// TIA Portal V18 export
FUNCTION_BLOCK "Pallets_Transport_System"   // FB9, LAD
{ S7_Optimized_Access := 'TRUE' }
// stored: MemoryReserve 100, SetENOAutomatically false
   VAR
      NumberOfPallet { S7_SetPoint := 'True'} : Int;
      Map : Array[1..4, 1..12] of Bool;
      MoveDirection : Int;   // 1-L, 2-Up, 3-R, 4-Down
      FoundSelectedPallet : Bool;
      CanMove : Bool;
   END_VAR
   VAR_TEMP
      i : Int;
      j : Int;
      k : Int;
   END_VAR
BEGIN

REGION Network 1 (SCL)
   // Sprawdzenie, które elementy sa wybrane i nadanie im nowej pozycji
   FOR #k := 1 TO 24 DO
       IF "Pallets_Stations".Pallets[#k].IsSelected THEN
           EXIT;
       END_IF;

   END_FOR;

   FOR #i := 1 TO 4 DO
       FOR #j := 1 TO 12 DO
           IF "Pallets_Stations".Pallets[#k].IsSelected THEN

               "Pallets_Stations".Pallets[#k].Station_Next_Position := "Pallets_Stations".Pallets[#k].Station_Current_Position;  // Initialisation

               CASE #MoveDirection OF
                   1:
                       IF "Pallets_Stations".Pallets[#k].Station_Next_Position[2] > 1 THEN  // Check Left
                           "Pallets_Stations".Pallets[#k].Station_Next_Position[2] := "Pallets_Stations".Pallets[#k].Station_Next_Position[2] - 1;
                       ELSE
                           #CanMove := FALSE;
                       END_IF;
                   3:
                       IF ("Pallets_Stations".Pallets[#k].Station_Next_Position[2] < 12) AND // Check Right
                           (("Pallets_Stations".Pallets[#k].Station_Next_Position[1] = 2 AND "Pallets_Stations".Pallets[#k].Station_Next_Position[2] < 12) OR ("Pallets_Stations".Pallets[#k].Station_Next_Position[1] <> 2 AND "Pallets_Stations".Pallets[#k].Station_Next_Position[2] < 11)) THEN
                           "Pallets_Stations".Pallets[#k].Station_Next_Position[2] := "Pallets_Stations".Pallets[#k].Station_Next_Position[2] + 1;
                       ELSE
                           #CanMove := FALSE;
                       END_IF;
                   2:
                       IF ("Pallets_Stations".Pallets[#k].Station_Next_Position[2] = 1) OR
                           (("Pallets_Stations".Pallets[#k].Station_Next_Position[1] = 1 AND "Pallets_Stations".Pallets[#k].Station_Next_Position[2] = 11) OR
                           ("Pallets_Stations".Pallets[#k].Station_Next_Position[1] = 2 AND "Pallets_Stations".Pallets[#k].Station_Next_Position[2] = 12) OR
                           ("Pallets_Stations".Pallets[#k].Station_Next_Position[1] = 3 AND "Pallets_Stations".Pallets[#k].Station_Next_Position[2] = 11) OR
                           ("Pallets_Stations".Pallets[#k].Station_Next_Position[1] = 4 AND "Pallets_Stations".Pallets[#k].Station_Next_Position[2] = 11)) THEN
                           IF "Pallets_Stations".Pallets[#k].Station_Next_Position[1] > 1 THEN
                               // Ruch w ostatniej kolumnie
                               IF "Pallets_Stations".Pallets[#k].Station_Next_Position[1] = 2 AND "Pallets_Stations".Pallets[#k].Station_Next_Position[2] = 12 THEN
                                   "Pallets_Stations".Pallets[#k].Station_Next_Position[1] := 1;
                                   "Pallets_Stations".Pallets[#k].Station_Next_Position[2] := 11;
                               ELSE
                                   "Pallets_Stations".Pallets[#k].Station_Next_Position[1] := "Pallets_Stations".Pallets[#k].Station_Next_Position[1] - 1;
                               END_IF;
                           ELSE
                               #CanMove := FALSE;
                           END_IF;
                       ELSE
                           #CanMove := FALSE;
                       END_IF;
                   4:
                       IF ("Pallets_Stations".Pallets[#k].Station_Next_Position[2] = 1) OR
                           (("Pallets_Stations".Pallets[#k].Station_Next_Position[1] = 1 AND "Pallets_Stations".Pallets[#k].Station_Next_Position[2] = 11) OR
                           ("Pallets_Stations".Pallets[#k].Station_Next_Position[1] = 2 AND "Pallets_Stations".Pallets[#k].Station_Next_Position[2] = 12) OR
                           ("Pallets_Stations".Pallets[#k].Station_Next_Position[1] = 3 AND "Pallets_Stations".Pallets[#k].Station_Next_Position[2] = 11) OR
                           ("Pallets_Stations".Pallets[#k].Station_Next_Position[1] = 4 AND "Pallets_Stations".Pallets[#k].Station_Next_Position[2] = 11)) THEN
                           IF "Pallets_Stations".Pallets[#k].Station_Next_Position[1] < 4 THEN
                               // Ruch w ostatniej kolumnie
                               IF "Pallets_Stations".Pallets[#k].Station_Next_Position[1] = 1 AND "Pallets_Stations".Pallets[#k].Station_Next_Position[2] = 11 THEN
                                   "Pallets_Stations".Pallets[#k].Station_Next_Position[1] := 2;
                                   "Pallets_Stations".Pallets[#k].Station_Next_Position[2] := 12;
                               ELSE
                                   "Pallets_Stations".Pallets[#k].Station_Next_Position[1] := "Pallets_Stations".Pallets[#k].Station_Next_Position[1] + 1;
                               END_IF;
                           ELSE
                               #CanMove := FALSE;
                           END_IF;
                       ELSE
                           #CanMove := FALSE;
                       END_IF;
               END_CASE;


               //TO DO Movement


               IF "Pallets_Stations".Stations["Pallets_Stations".Pallets[#k].Station_Next_Position[1], "Pallets_Stations".Pallets[#k].Station_Next_Position[2]].IsEmpty THEN
                   // Aktualizacja stanu stanowisk i palet


                   // Aktualizacja pozycji palety
                   "Pallets_Stations".Pallets[#k].Station_Current_Position := "Pallets_Stations".Pallets[#k].Station_Next_Position;
                   #CanMove := TRUE;
               ELSE
                   #CanMove := FALSE;  // Nowe stanowisko zajęte
               END_IF;


           END_IF;
       END_FOR;
   END_FOR;
END_REGION
END_FUNCTION_BLOCK
